{attribute 'GeneratedUsingTerminal: EL7411-0000-0016'}
{attribute addProperty BoxType "EL7411-0000-0016"}
{attribute addProperty Id "Target_positionAT %Q*UDINT4"}
{attribute addProperty CRC "86249236"}
{attribute addProperty Size "4"}
TYPE DRV_Target_position_05240F14 :
STRUCT
	{attribute addProperty Name "Target_position"}
	Target_position AT %Q* : UDINT;
END_STRUCT
END_TYPE

(* stored: Version 1.2.0.0, ProductVersion 3.1.4024.9
   DUT DRV_Target_position_05240F14: Id {7c38b7e5-04ed-4a76-b004-91028a4eaaa5} *)
